TYPE ST_ScrewdriverCommand :
STRUCT
    bPcControl : BOOL;
    bTighten   : BOOL;
    bLoosen    : BOOL;
    bStop      : BOOL;
    bReset     : BOOL;
END_STRUCT
END_TYPE

(* stored: Version 1.1.0.1, ProductVersion 3.1.4026.20
   DUT ST_ScrewdriverCommand: Id {1C8FF05D-48F7-4561-A89A-201364774812} *)
